Universal Robots PolyScope program: mecspe_refactor.urp

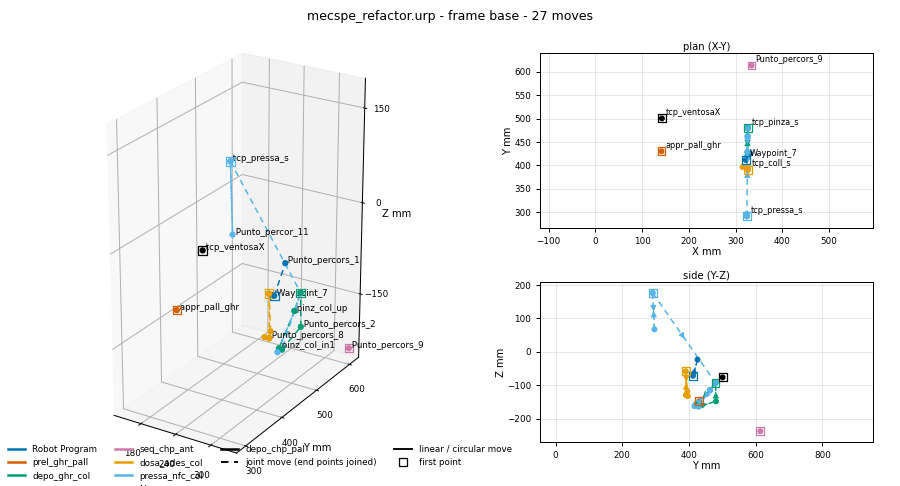
[picture p0: tool path of mecspe_refactor.urp in frame base, 27 of 40 moves have a stored position in this frame; points joined in program order, loops and branches not executed]
Program mecspe_refactor (installation=mecspe_install directory=/home/ur/ursim-current/programs/mecspe2 createdIn=3.15.4.106291 lastSavedIn=3.15.4.106291 robotSerialNumber=2018359999)
Calibrated DH parameters: a=[0.000104, -0.381245, -0.385946, 0.00002, 0.000083, 0]; d=[0.089177, 59.99214, -36.297918, -23.584132, 0.094784, 0.082552]; alpha=[1.570197, -0.003145, 0.002952, 1.570494, -1.570091, 0]; deltaTheta=[-0.00001, -0.459739, 0.638868, -0.17972, -0.000006, -0.000462]
InitVariablesNode variables(variable(name=ghr, expression=2), variable(name=nCycle, expression=0), variable(name=pallStocks, expression=[16,16,16,40,16,16,16,40,16,16,16,40,16,40,0,0,0,0,0,0,0,0,0,0]), variable(name=pick, expression=[0,0]))
BeforeStart
  Script file /home/ur/ursim-current/programs/mecspe2/calc_pose_to_position.script
    | def calc_pose_to_position(pose, feature, position):
    | 
    |    PoseRelativeToFeature = pose_trans(pose_inv(feature), pose)
    | 
    |    diff = pose_sub(position, PoseRelativeToFeature)
    |    vect = p[diff[0], diff[1], diff[2], 0, 0, 0]
    | 
    |    MoveTCPRelativeToFeature = pose_add(PoseRelativeToFeature, vect)
    |    return pose_trans(feature, MoveTCPRelativeToFeature)
    | 
    | end
  Script file /home/ur/ursim-current/programs/mecspe2/calc_item_position.script
    | def calc_item_position(item, prop, grid, module, seat, compens):
    | 
    |     # calcola la posizione assoluta del pezzo scelto da pickPalletItem
    | 
    |     # nPosX è il numero di colonne
    |     # nPosY è il numero di righe
    |     # distX è la distanza tra colonne
    |     # distY è la distanza tra righe
    |     # [posX1, posY1] è la posizione del primo pezzo rispetto all'origine del pallet
    | 
    |     nPallet = module # module e seat partono da 1
    |     nItem = seat
    | 
    |     nPosXgrid = grid[0] # numero di posizioni della giglia in X
    |     distXgrid = grid[2] # distanza tra gli slot della griglia in X
    |     distYgrid = grid[3] # distanza tra gli slot della griglia in Y
    | 
    |     pallPosX = nPallet%nPosXgrid
    |     if(pallPosX==0): pallPosX = nPosXgrid end
    |     pallPosY = ceil(nPallet/nPosXgrid)
    | 
    |     pallPosX1 = grid[4]
    |     pallPosY1 = grid[5]
    | 
    | 
    |     nPosX = prop[item,0]
    |     nPosY = prop[item,1]
    |     distX = prop[item,2]
    |     distY = prop[item,3]
    |     posX1 = prop[item,4]
    |     posY1 = prop[item,5]
    | 
    |     posX = nItem%nPosX
    |     if(posX==0): posX = nPosX end
    |     posY = ceil(nItem/nPosX)
    | 
    |     position = p[0,0,0,0,0,0]
    | 
    |     X=distX*(posX - 1) + posX1 + distXgrid*(pallPosX - 1) + pallPosX1 + compens[0]*1000
    |     Y=distY*(posY - 1) + posY1 + distYgrid*(pallPosY - 1) + pallPosY1 + compens[1]*1000
    | 
    |     position[0] = X/1000
    |     position[1] = Y/1000
    | 
    |     return position
    | 
    |  end
  Script file /home/ur/ursim-current/programs/mecspe2/calc_compens_pos.script
    | def calc_compens_pos(item, prop, grid, module, feature, posAppr):
    | 
    | 	compens = p[0,0,0,0,0,0]
    | 	posPred = calc_item_position(item, prop, grid, module, 1, compens)
    | 
    | 	posApprFeat = pose_trans(pose_inv(feature), posAppr)
    | 	diff = pose_sub(posApprFeat - posPred)
    | 
    | 	compens[0] = diff[0]
    | 	compens[1] = diff[1]
    | 
    | 	return compens
    | 
    | end
  Script file /home/ur/ursim-current/programs/mecspe2/tcpMov.script
    | def tcpMov(vect):
    | 
    |     # FeaturePose is the pose for the feature
    |     # vect = p[0.1, 0, 0, 0, 0, 0] makes us move 10cm in the X direction of the feature
    |     # credits: https://forum.universal-robots.com/t/move-tcp-relative-to-feature/15492
    | 
    |    tcp_pose = get_actual_tcp_pose()
    |    return pose_add(tcp_pose, vect)
    | 
    | 
    | end
  Script file /home/ur/ursim-current/programs/mecspe2/gen_tcp_grid.script
    | def next_tcp_grid_pos(cur_pos,size,dist):
    | 
    | # size e' la dimensione della griglia da generare,
    | # 2 significa 2x2, 3 significa 3x3 etc
    | 
    | rel_p = [0,0]
    | tcpp = get_actual_tcp_pose()
    | 
    | posX = cur_pos%size
    | if(posX==0): posX = size end
    | posY = ceil(cur_pos/size)
    | 
    | actual_dx = -dist*(size-1)/2 + (posX-1)*dist
    | actual_dy= -dist*(size-1)/2 + (posY-1)*dist
    | 
    | posX = (cur_pos+1)%size
    | if(posX==0): posX = size end
    | posY = ceil((cur_pos+1)/size)
    | 
    | next_dx = -dist*(size-1)/2 + (posX-1)*dist
    | next_dy= -dist*(size-1)/2 + (posY-1)*dist
    | 
    | rel_p = [next_dx - actual_dx, next_dy - actual_dy]
    | 
    | return rel_p
    | 
    | end
  Script file /home/ur/ursim-current/programs/andrea11/stockUpdate.script_bak
    | def stockUpdate(pick,stock):
    | 
    |     # simple function that ingests the output of pickItem and returns the
    |     # modified stock array. just so to avoid using global variables and
    |     # multi-dimensional arrays
    | 
    |     i = pick[0]
    |     stock[i] = stock[i] - 1
    |     return stock
    | 
    | 
    | end
  Script file /home/ur/ursim-current/programs/mecspe2/pickPalletItem.script
    | def pickPalletItem(type, pallDefs, pallTypes, pallStocks):
    | 
    |   # seleziona un pezzo sulla griglia, noti il tipo di pezzo e lo stato della griglia
    | 
    |   # lo script funziona finché le variabili del robot non vengono resettate. Tuttavia, anche
    |   # in caso di riavvio, è possibile scrivere manualmente le info sulla griglia e lo stock
    |   # all'inizio del programma, così da 'insegnare' al robot dove farlo
    |   # riprendere
    | 
    |   iPallet = 0 # inizializzo l'id del pallet
    | 
    |   while iPallet < length(pallStocks):
    | 
    |     if pallTypes[iPallet] == type and pallStocks[iPallet] > 0 :
    | 
    |       nItems = pallStocks[iPallet] # numero di pezzi nello stock del pallet iesimo
    | 
    |       nPosX = pallDefs[type,0] # numero di posizioni lungo x, come definito per il pallet di tipo "type"
    |       nPosY = pallDefs[type,1] # numero di posizioni lungo y, come definito per il pallet di tipo "type"
    | 
    |       stockMax = nPosX*nPosY
    |       iItem = stockMax - nItems # id del pezzo
    | 
    |       pick = [iPallet,iItem]
    | 
    |       # pick = [id del pallet, id del pezzo]
    | 
    |       return pick
    |  end
    | iPallet = iPallet + 1
    | end
    | end
  Script file /home/ur/ursim-current/programs/mecspe2/ini_grid.script
    | def ini_grid():
    | 
    |     # grid = [nPallPosX, nPallPosY, distPallX, distPallY, pallPosX1, pallPosY1, pallPosZ1]
    |     # la struttura e' del tutto analoga in logica con quella espressa in defs
    |     grid = [4, 6, 90, 90, 10, 20, 6]
    |     return grid
    | end
  Script file /home/ur/ursim-current/programs/mecspe2/ini_defs.script
    | chp = 1
    | ghr = 2
    | 
    | def ini_defs():
    | 
    |     # definition = [nPosX,nPosY,distX,distY,posX1,posY1,posZ1]
    | 
    |     # nPosX è il numero di colonne
    |     # nPosY è il numero di righe
    |     # distX è la distanza tra colonne
    |     # distY è la distanza tra righe
    |     # [posX1, posY1] è la posizione del primo pezzo rispetto all'origine del pallet
    |     # posZ1 e' la posizione che deve raggiungere il TCP lungo asse Z, che sarebbe asse verticale
    | 
    |     defs = [
    |         [0, 0, 0, 0, 0, 0, 0], # slot vuoto
    |         [4, 10, 18, 8, 17, 10.3, 10], # pallet chip
    |         [4, 4, 21, 21, 12.5, 12.5, 50], # pallet ghiere
    |         [1, 1, 0, 0, 132.06, 44, 16.05], # stazione antenna
    |         [1, 2, 0, 40, 20.256, 24, 27.85], # stazione incollaggio
    |         [1, 1, 0, 0, 40, 40, 50] # cestino
    |     ]
    |     return defs
    | end
  Script file /home/ur/ursim-current/programs/mecspe2/ini_types.script_bak_bak
    | def ini_types():
    | 
    |     visualTypes = [
    | 
    |         [0, 0, 0, 0],
    |         [0, 0, 0, 0],
    |         [0,0,0,0],
    |         [0,0,0,0],
    |         [0,ghr,0,chp],
    |         [0,0,0,0]
    | 
    |     ]
    | 
    | # purtroppo fare questa array vuota di dimensione (righe)x(colonne) per aggirare le limitazioni di UR
    | # bisogna ricordarsi di cambiare questa dichiarazione di types se si cambia dimensione griglia
    | 
    |      types = [0,0,0,0,0,0,0,0,0,0,0,0,0,0,0,0,0,0,0,0,0,0,0,0]
    | 
    |     iii = 0
    |     s = size(visualTypes)
    |     i = 0
    |     while i < s[0]:
    | 
    |         ii=0
    |         while ii < s[1]:
    | 
    |             types[iii] = visualTypes[s[0]-1-i,ii]
    |             ii = ii + 1
    |             iii = iii + 1
    |         end
    |     i = i + 1
    |     end
    |     return types
    | end
  Script file /home/ur/ursim-current/programs/mecspe2/ini_stocks.script
    | def ini_stocks(defs, types):
    | 
    |     global f = -1 # usa questo carattere per inizializzare automaticamente pallet pieni
    | 
    |     visualStocks = [
    | 
    |         [f, f, f, f],
    |         [f, f, f, f],
    |         [f, f, f, f],
    |         [f, f, f, f],
    |         [f, f, f, f],
    |         [f ,f, f, f]
    | 
    |     ]
    | 
    | # purtroppo occorre fare questa array vuota di dimensione (righe)x(colonne) per aggirare le limitazioni di UR
    | # bisogna ricordarsi di cambiare questa dichiarazione di types se si cambia dimensione griglia
    | 
    |      stocks = [0,0,0,0,0,0,0,0,0,0,0,0,0,0,0,0,0,0,0,0,0,0,0,0]
    | 
    |     iii = 0
    |     s = size(visualStocks)
    |     i = 0
    |     while i < s[0]:
    | 
    |         ii=0
    |         while ii < s[1]:
    |             if visualStocks[s[0]-1-i,ii] == f:
    |                 nPosX = defs[types[iii], 0]
    |                 nPosY = defs[types[iii], 1]
    |                 stocks[iii] = nPosX*nPosY
    |             else:
    | 
    |                 stocks[iii] = visualStocks[s[0]-1-i,ii]
    |             end
    |             ii = ii + 1
    |             iii = iii + 1
    |         end
    |     i = i + 1
    |     end
    |     return stocks
    | end
  Script file /home/ur/ursim-current/programs/mecspe2/fun_tens_utensile.script
    | def fun_tens_utensile():
    | 
    | 	i = 0
    | 	# invia 3 "impulsi" alla macchina per assicurarsi che il tool abbia tensione
    | 	while i < 3:
    | 		set_tool_voltage(24)
    | 		sleep(0.24)
    | 		i = i + 1
    | 	end
    | 
    | end
  posApproccio := get_actual_tcp_pose()
  statoPinza := 0
  statoGhiera := 0
  statoChip := 0
  compens := p[0,0,0,0,0,0]
  Set DigitalOutput pin=DO_ventosaOff; digitalValue=1
  Set DigitalOutput pin=DO_ventosaOn; digitalValue=0
  Set DigitalOutput pin=digital_out[2]; digitalValue=0
  pallTypes := ini_types()
  bypassVerifChp := False
  grid := ini_grid()
  pallDefs := ini_defs()
  pallStocks := ini_stocks(pallDefs,pallTypes)
  nCycle := 1
  chp_check := False
  Script: fun_tens_utensile()
  Wait Sleep waitTime=1
Robot Program (runOnlyOnce=false)
  MoveJ speed 60 deg/s, acceleration 80 deg/s^2 (useActiveTCP=true)
    Waypoint Waypoint_7: TCP in base x=321.623 y=412.075 z=-71.725 mm, rx=1.5831 ry=-2.4822 rz=0.1268 rad; joints [-138.339, -65.21, 105.073, -118.045, -93.062, 36.92] deg; flange x=345.08 y=447.244 z=123.756 mm, rx=2.1618 ry=-1.9789 rz=0.0478 rad
  Timer (action=Start) variable(name=timer_1)
  apprendimento := True
  item := ghr
  pick := pickPalletItem(item,pallDefs,pallTypes,pallStocks)
  lastpick := pick
  Call prel_ghr_pall
  statoGhiera := 1
  Call depo_ghr_col
  statoGhiera := 2
  chp_check := False
  Loop While (checkContinuously=false) expression=chp_check≟ False
    item := chp
    pick := pickPalletItem(item,pallDefs,pallTypes,pallStocks)
    Call prel_chp_pall
    statoChip := 1
    pallStocks := stockUpdate(pick,pallStocks)
    MoveJ speed 60 deg/s, acceleration 80 deg/s^2 (useActiveTCP=false) tcp=Ventosa
      Waypoint Punto_percors_1: TCP in base x=331.541 y=425.449 z=-23.301 mm, rx=1.7621 ry=-0.7398 rz=-1.7726 rad; joints [-145.076, -38.163, 77.174, -38.938, -53.96, -45.259] deg; flange x=377.019 y=458.221 z=10.448 mm, rx=1.7621 ry=-0.7398 rz=-1.7726 rad
    Call seq_chp_ant
    If chp_check≟ True
      Call dosa_ades_col
      Call pressa_nfc_col
      Call prel_ghr_col
    Else 
      Call depo_chp_pal
Thread Thread_1 (runOnlyOnce=false)
  If timer_1>4
    Timer (action=Reset) variable=timer_1
    Script: fun_tens_utensile()
    Timer (action=Start) variable=timer_1
SubProgram -> prel_ghr_pall
SubProgram  [hidden by the author, left out]
SubProgram  [hidden by the author, left out]
SubProgram depo_ghr_pall [hidden by the author, left out]
SubProgram -> depo_chp_pal
SubProgram -> seq_chp_ant
SubProgram -> depo_ghr_col
SubProgram -> dosa_ades_col
SubProgram -> pressa_nfc_col
SubProgram prel_ghr_pall (keepSynchronizedWithDisk=false)
  If apprendimento≟ True
    MoveJ speed 60 deg/s, acceleration 80 deg/s^2 (useActiveTCP=false) tcp=Pinza
      Waypoint appr_pall_ghr: TCP in base x=141.508 y=430.186 z=-147.75 mm, rx=0.607 ry=-1.4882 rz=-0.6293 rad; joints [-125.755, -39.244, 81.167, -41.963, -34.571, 44.831] deg; flange x=189.515 y=570.182 z=1.456 mm, rx=0.607 ry=-1.4882 rz=-0.6293 rad
      modulo :=  (valueSource=Operator message=Specificare il numero di modulo usato per l'apprendimento valueType=Integer)
  Else 
    MoveJ speed 60 deg/s, acceleration 80 deg/s^2 (useActiveTCP=false) tcp=Pinza
      Script: posApproccio = pose_trasf(posa, riferimento, vettore)
      Waypoint Waypoint (Variable): variable=posApproccio
  MoveL speed 250 mm/s, acceleration 1200 mm/s^2 (useActiveTCP=false) tcp=Pinza; feature=Base
    Waypoint Waypoint_1 (Relative): relativeFromPosition TCP in base x=143.961 y=537.139 z=34.835 mm, rx=0.607 ry=-1.4882 rz=-0.6293 rad; joints [-125.506, -39.287, 81.209, -42.035, -34.619, 44.824] deg; TCP in base x=143.457 y=501.955 z=-0.687 mm, rx=0.607 ry=-1.4882 rz=-0.6293 rad; joints [-127.449, -38.931, 87.822, -48.999, -36.562, 44.817] deg; flange x=189.012 y=534.998 z=-34.066 mm, rx=0.607 ry=-1.4882 rz=-0.6293 rad
  MoveL speed 50 mm/s, acceleration 100 mm/s^2 (useActiveTCP=false) tcp=Pinza; feature=Base
    Waypoint Waypoint_2 (Relative): relativeFromPosition TCP in base x=143.457 y=501.955 z=-0.687 mm, rx=0.607 ry=-1.4882 rz=-0.6293 rad; joints [-127.449, -38.931, 87.822, -48.999, -36.562, 44.817] deg; TCP in base x=143.286 y=489.992 z=-12.765 mm, rx=0.607 ry=-1.4882 rz=-0.6293 rad; joints [-128.156, -38.626, 89.864, -51.344, -37.269, 44.815] deg; flange x=188.841 y=523.035 z=-46.144 mm, rx=0.607 ry=-1.4882 rz=-0.6293 rad
    SuppressedNode
      Script: tool()
    Waypoint Waypoint_3 (Relative): relativeFromPosition TCP in base x=143.286 y=489.992 z=-12.765 mm, rx=0.607 ry=-1.4882 rz=-0.6293 rad; joints [-128.156, -38.626, 89.864, -51.344, -37.269, 44.815] deg; TCP in base x=143.457 y=501.955 z=-0.687 mm, rx=0.607 ry=-1.4882 rz=-0.6293 rad; joints [-127.449, -38.931, 87.822, -48.999, -36.562, 44.817] deg; flange x=189.012 y=534.998 z=-34.066 mm, rx=0.607 ry=-1.4882 rz=-0.6293 rad
  MoveL speed 250 mm/s, acceleration 1200 mm/s^2 (useActiveTCP=false) tcp=Pinza; feature=Base
    Waypoint Waypoint_4 (Relative): relativeFromPosition TCP in base x=143.457 y=501.955 z=-0.687 mm, rx=0.607 ry=-1.4882 rz=-0.6293 rad; joints [-127.449, -38.931, 87.822, -48.999, -36.562, 44.817] deg; TCP in base x=143.961 y=537.139 z=34.835 mm, rx=0.607 ry=-1.4882 rz=-0.6293 rad; joints [-125.506, -39.287, 81.209, -42.035, -34.619, 44.824] deg; flange x=189.515 y=570.182 z=1.456 mm, rx=0.607 ry=-1.4882 rz=-0.6293 rad
SubProgram depo_ghr_col (keepSynchronizedWithDisk=false)
  MoveJ speed 60 deg/s, acceleration 80 deg/s^2 (useActiveTCP=false) tcp=Pinza
    Waypoint tcp_pinza_s: TCP in base x=326.011 y=479.267 z=-92.696 mm, rx=0.6076 ry=-1.4868 rz=-0.6287 rad; joints [-134.797, -24.75, 41.969, -17.153, -43.759, 44.739] deg; flange x=373.998 y=619.302 z=56.479 mm, rx=0.6076 ry=-1.4868 rz=-0.6287 rad
    Waypoint pinz_col_up: TCP in base x=325.773 y=462.541 z=-115.349 mm, rx=-0.2128 ry=-1.5595 rz=0.1908 rad; joints [-132.675, 4.221, 14.51, -18.717, -41.716, 104.821] deg; flange x=376.545 y=660.076 z=-162.724 mm, rx=-0.2162 ry=-1.5589 rz=0.1901 rad
    Waypoint pinz_col_in1: TCP in base x=325.228 y=420.094 z=-158.165 mm, rx=-0.2127 ry=-1.5596 rz=0.1906 rad; joints [-134.83, -0.501, 31.804, -31.303, -43.826, 104.834] deg; flange x=374.048 y=618.963 z=-205.428 mm, rx=-0.2127 ry=-1.5596 rz=0.1906 rad
    SuppressedNode
      URCap Close Gripper (SCHUNK End-of-Arm Modular System for UR, SCHUNK GmbH & Co.)
    Waypoint pinz_col_out: TCP in base x=325.373 y=428.559 z=-163.725 mm, rx=-0.2126 ry=-1.5596 rz=0.1907 rad; joints [-134.386, 1.907, 27.313, -29.22, -43.4, 104.831] deg; flange x=374.171 y=627.435 z=-210.98 mm, rx=-0.2126 ry=-1.5596 rz=0.1907 rad
    SuppressedNode
      Waypoint pinz_col_up: TCP in base x=353.537 y=408.471 z=-60.29 mm, rx=1.9378 ry=-1.1643 rz=-1.0825 rad; joints [-133.591, -22.853, 54.464, -66.388, -55.09, 0.038] deg; flange x=383.886 y=633.812 z=-67.559 mm, rx=1.9378 ry=-1.1643 rz=-1.0825 rad
    Waypoint Punto_percors_2: TCP in base x=326.04 y=480.901 z=-148.453 mm, rx=0.4029 ry=-1.5348 rz=-0.4259 rad; joints [-133.017, -11.499, 29.335, -17.8, -41.967, 59.778] deg; flange x=376.733 y=653.438 z=-40.877 mm, rx=0.3991 ry=-1.5354 rz=-0.4274 rad
    SuppressedNode
      URCap Open Gripper (SCHUNK End-of-Arm Modular System for UR, SCHUNK GmbH & Co.)
    Waypoint tcp_pinza_s: TCP in base x=326.011 y=479.267 z=-92.696 mm, rx=0.6076 ry=-1.4868 rz=-0.6287 rad; joints [-134.797, -24.75, 41.969, -17.153, -43.759, 44.739] deg; flange x=373.998 y=619.302 z=56.479 mm, rx=0.6076 ry=-1.4868 rz=-0.6287 rad
SubProgram prel_chp_pall [hidden by the author, left out]
SubProgram seq_chp_ant (keepSynchronizedWithDisk=false)
  If apprendimento≟ True
    MoveJ speed 60 deg/s, acceleration 80 deg/s^2 (useActiveTCP=false) tcp=Ventosa
      Waypoint Punto_percors_9: TCP in base x=334.202 y=613.623 z=-237.914 mm, rx=1.7619 ry=-0.7398 rz=-1.7727 rad; joints [-133.692, 7.188, 14.603, -21.767, -42.719, -45.183] deg; flange x=379.684 y=646.401 z=-204.176 mm, rx=1.7619 ry=-0.7398 rz=-1.7727 rad
  Else 
    MoveJ speed 60 deg/s, acceleration 80 deg/s^2 (useActiveTCP=false) tcp=Pinza
      SuppressedNode
        Script: pos_approccio = calc_rel_pose()
      Waypoint Waypoint (Variable): variable=posApproccio
  MoveL speed 50 mm/s, acceleration 100 mm/s^2 (useActiveTCP=false) tcp=Ventosa; feature=Base
    Waypoint Waypoint_5 (Relative): relativeFromPosition TCP in base x=334.202 y=613.623 z=-237.914 mm, rx=1.7619 ry=-0.7398 rz=-1.7727 rad; joints [-133.509, 7.247, 14.462, -21.694, -42.684, -45.282] deg; TCP in base x=333.934 y=593.03 z=-258.697 mm, rx=1.762 ry=-0.7397 rz=-1.7726 rad; joints [-134.549, 4.522, 23.777, -28.293, -43.727, -45.281] deg; flange x=379.412 y=625.807 z=-224.951 mm, rx=1.762 ry=-0.7397 rz=-1.7726 rad
    If bypassVerifChp≟ True
      chp_check := True
    ElseIf digital_in[0]≟ False
      chp_check :=  (valueSource=Operator message=L'antenna nfc non risponde. Si prega di confermare la funzionalita' del sensore valueType=Boolean)
    Else 
      Loop Counting (count=5) loopVariable(name=Loop_1)
        Wait Sleep waitTime=0.5
        If DI_chpVerif≟ True
          chp_check := True
    Waypoint Waypoint_6 (Relative): relativeFromPosition TCP in base x=333.934 y=593.03 z=-258.697 mm, rx=1.762 ry=-0.7397 rz=-1.7726 rad; joints [-134.549, 4.522, 23.777, -28.293, -43.727, -45.281] deg; TCP in base x=334.202 y=613.623 z=-237.914 mm, rx=1.7619 ry=-0.7398 rz=-1.7727 rad; joints [-133.509, 7.247, 14.462, -21.694, -42.684, -45.282] deg; flange x=379.684 y=646.401 z=-204.176 mm, rx=1.7619 ry=-0.7398 rz=-1.7727 rad
SubProgram dosa_ades_col (keepSynchronizedWithDisk=false)
  MoveJ speed 60 deg/s, acceleration 80 deg/s^2 (useActiveTCP=false) tcp=Dosatore_Colla
    Waypoint tcp_coll_s: TCP in base x=326.049 y=390.336 z=-58.733 mm, rx=1.5073 ry=-2.6452 rz=0.2028 rad; joints [-138.926, -70.014, 111.07, -124.336, -96.301, 42.443] deg; flange x=328.586 y=422.248 z=138.688 mm, rx=2.1203 ry=-2.1445 rz=0.1587 rad
    Waypoint Punto_percors_7: TCP in base x=326.117 y=395.016 z=-120.075 mm, rx=1.5072 ry=-2.6453 rz=0.2028 rad; joints [-138.56, -63.27, 112.967, -132.934, -96.298, 42.835] deg; flange x=328.653 y=426.927 z=77.346 mm, rx=2.1202 ry=-2.1446 rz=0.1587 rad
    Waypoint Punto_percors_8: TCP in base x=326.087 y=391.561 z=-129.594 mm, rx=1.5073 ry=-2.6453 rz=0.2028 rad; joints [-138.834, -62.452, 113.712, -134.529, -96.337, 42.56] deg; flange x=328.619 y=423.469 z=67.828 mm, rx=2.1203 ry=-2.1446 rz=0.1587 rad
  MoveL speed 250 mm/s, acceleration 1200 mm/s^2 (useActiveTCP=false) tcp=Dosatore_Colla; feature=Base
    Waypoint Punto_percors_8: TCP in base x=326.087 y=391.561 z=-129.594 mm, rx=1.5073 ry=-2.6453 rz=0.2028 rad; joints [-138.834, -62.452, 113.712, -134.529, -96.337, 42.56] deg; flange x=328.619 y=423.469 z=67.828 mm, rx=2.1203 ry=-2.1446 rz=0.1587 rad
    Waypoint arco01: TCP in base x=314.98 y=396.61 z=-132.865 mm, rx=-1.4222 ry=2.3645 rz=-0.9681 rad; joints [-120.617, -54.723, 114.843, -141.201, -129.749, 60.945] deg; flange x=216.441 y=481.445 z=19.098 mm, rx=-2.0946 ry=2.021 rz=-1.0736 rad
    Set DigitalOutput pin=digital_out[2]; digitalValue=1
    Wait Sleep waitTime=0.5
    Waypoint Punto_percors_8: TCP in base x=326.087 y=391.561 z=-129.594 mm, rx=1.5073 ry=-2.6453 rz=0.2028 rad; joints [-138.834, -62.452, 113.712, -134.529, -96.337, 42.56] deg; flange x=328.619 y=423.469 z=67.828 mm, rx=2.1203 ry=-2.1446 rz=0.1587 rad
    Set DigitalOutput pin=digital_out[2]; digitalValue=0
  MoveJ speed 60 deg/s, acceleration 80 deg/s^2 (useActiveTCP=false) tcp=Dosatore_Colla
    Waypoint tcp_coll_s: motionParameters(blendRadius=0.005); TCP in base x=326.049 y=390.336 z=-58.733 mm, rx=1.5073 ry=-2.6452 rz=0.2028 rad; joints [-138.926, -70.014, 111.07, -124.336, -96.301, 42.443] deg; flange x=328.586 y=422.248 z=138.688 mm, rx=2.1203 ry=-2.1445 rz=0.1587 rad
SubProgram pressa_nfc_col (keepSynchronizedWithDisk=false)
  MoveJ speed 60 deg/s, acceleration 80 deg/s^2 (useActiveTCP=false) tcp=Pressa
    SuppressedNode
      Waypoint tcp_ventosaY_s: TCP in base x=355.984 y=389.916 z=-58.857 mm, rx=-1.401 ry=-1.0647 rz=1.3858 rad; joints [-146.472, -36.177, 73.345, -37.097, -55.375, 194.745] deg; flange x=401.93 y=456.119 z=8.64 mm, rx=-1.401 ry=-1.0647 rz=1.3858 rad
    Waypoint tcp_pressa_s: TCP in base x=324.299 y=291.031 z=176.511 mm, rx=-1.4012 ry=-1.0643 rz=1.3857 rad; joints [-148.69, -46.659, 85.022, -38.277, -57.561, -165.274] deg; flange x=370.992 y=407.578 z=60.385 mm, rx=-1.4012 ry=-1.0643 rz=1.3857 rad
    Waypoint Punto_percor_11: TCP in base x=324.225 y=296.228 z=67.341 mm, rx=-1.3969 ry=-1.0517 rz=1.3843 rad; joints [-148.364, -36.011, 84.683, -48.026, -56.743, -165.537] deg; flange x=370.899 y=412.4 z=-49.168 mm, rx=-1.3969 ry=-1.0517 rz=1.3843 rad
    Wait Sleep waitTime=5
    Waypoint tcp_pressa_s: TCP in base x=324.299 y=291.031 z=176.511 mm, rx=-1.4012 ry=-1.0643 rz=1.3857 rad; joints [-148.69, -46.659, 85.022, -38.277, -57.561, -165.274] deg; flange x=370.992 y=407.578 z=60.385 mm, rx=-1.4012 ry=-1.0643 rz=1.3857 rad
  MoveJ speed 60 deg/s, acceleration 80 deg/s^2 (useActiveTCP=false) tcp=Pinza
    Waypoint tcp_pinza_s: TCP in base x=326.011 y=479.267 z=-92.696 mm, rx=0.6076 ry=-1.4868 rz=-0.6287 rad; joints [-134.797, -24.75, 41.969, -17.153, -43.759, 44.739] deg; flange x=373.998 y=619.302 z=56.479 mm, rx=0.6076 ry=-1.4868 rz=-0.6287 rad
    Waypoint pinz_col_up: TCP in base x=325.773 y=462.541 z=-115.349 mm, rx=-0.2128 ry=-1.5595 rz=0.1908 rad; joints [-132.675, 4.221, 14.51, -18.717, -41.716, 104.821] deg; flange x=376.545 y=660.076 z=-162.724 mm, rx=-0.2162 ry=-1.5589 rz=0.1901 rad
    Waypoint pinz_col_out: TCP in base x=325.373 y=428.559 z=-163.725 mm, rx=-0.2126 ry=-1.5596 rz=0.1907 rad; joints [-134.386, 1.907, 27.313, -29.22, -43.4, 104.831] deg; flange x=374.171 y=627.435 z=-210.98 mm, rx=-0.2126 ry=-1.5596 rz=0.1907 rad
    Waypoint pinz_col_in: TCP in base x=325.232 y=416.122 z=-162.784 mm, rx=-0.2125 ry=-1.5596 rz=0.1904 rad; joints [-135.043, -0.583, 32.776, -32.194, -44.036, 104.821] deg; flange x=374.053 y=615.003 z=-209.997 mm, rx=-0.2125 ry=-1.5596 rz=0.1904 rad
    SuppressedNode
      URCap Open Gripper (SCHUNK End-of-Arm Modular System for UR, SCHUNK GmbH & Co.)
    Waypoint pinz_col_up: TCP in base x=325.773 y=462.541 z=-115.349 mm, rx=-0.2128 ry=-1.5595 rz=0.1908 rad; joints [-132.675, 4.221, 14.51, -18.717, -41.716, 104.821] deg; flange x=376.545 y=660.076 z=-162.724 mm, rx=-0.2162 ry=-1.5589 rz=0.1901 rad
    SuppressedNode
      Waypoint pinz_col_up: TCP in base x=353.537 y=408.471 z=-60.29 mm, rx=1.9378 ry=-1.1643 rz=-1.0825 rad; joints [-133.591, -22.853, 54.464, -66.388, -55.09, 0.038] deg; flange x=383.886 y=633.812 z=-67.559 mm, rx=1.9378 ry=-1.1643 rz=-1.0825 rad
    SuppressedNode
      Waypoint Punto_percors_2: TCP in base x=354.064 y=441.822 z=-77.166 mm, rx=1.8482 ry=-1.2116 rz=-0.904 rad; joints [-131.419, -13.619, 42.947, -63.355, -59.194, 8.709] deg; flange x=380.052 y=663.563 z=-120.852 mm, rx=1.8482 ry=-1.2116 rz=-0.904 rad
    SuppressedNode
      URCap Open Gripper (SCHUNK End-of-Arm Modular System for UR, SCHUNK GmbH & Co.)
    Waypoint tcp_pinza_s: TCP in base x=326.011 y=479.267 z=-92.696 mm, rx=0.6076 ry=-1.4868 rz=-0.6287 rad; joints [-134.797, -24.75, 41.969, -17.153, -43.759, 44.739] deg; flange x=373.998 y=619.302 z=56.479 mm, rx=0.6076 ry=-1.4868 rz=-0.6287 rad
SubProgram prel_ghr_col [hidden by the author, left out]
SubProgram depo_chp_pal (keepSynchronizedWithDisk=false)
  If apprendimento≟ True
    MoveJ speed 60 deg/s, acceleration 80 deg/s^2 (useActiveTCP=false) tcp=Ventosa
      Waypoint tcp_ventosaX: TCP in base x=142.442 y=500.567 z=-76.685 mm, rx=1.7622 ry=-0.7397 rz=-1.7725 rad; joints [-127.721, -38.126, 88.043, -49.879, -36.592, -45.229] deg; flange x=187.914 y=533.343 z=-42.931 mm, rx=1.7622 ry=-0.7397 rz=-1.7725 rad
  Else 
    MoveJ speed 60 deg/s, acceleration 80 deg/s^2 (useActiveTCP=false) tcp=Pinza
      SuppressedNode
        Script: pos_approccio = calc_rel_pose()
      Waypoint Waypoint (Variable): variable=posApproccio
  MoveL speed 250 mm/s, acceleration 1000 mm/s^2 (useActiveTCP=false) tcp=Ventosa; feature=Base
    Waypoint Punto_percor_22 (Relative): relativeFromPosition TCP in base x=35.118 y=689.646 z=-262.532 mm, rx=1.7853 ry=-0.7339 rz=-1.771 rad; joints [-111.426, -3.8, 43.305, -41.846, -20.436, -43.809] deg; TCP in base x=33.407 y=563.018 z=-390.38 mm, rx=1.7855 ry=-0.7339 rz=-1.7712 rad; joints [-115.654, -0.107, 63.287, -65.282, -24.633, -44.07] deg; flange x=78.389 y=595.329 z=-355.54 mm, rx=1.7855 ry=-0.7339 rz=-1.7712 rad
  MoveL speed 100 mm/s, acceleration 100 mm/s^2 (useActiveTCP=false) tcp=Ventosa; feature=Base
    Set DigitalOutput pin=DO_ventosaOff; digitalValue=1
    Set DigitalOutput pin=digital_out[0]; digitalValue=0
    Waypoint Punto_percor_24 (Relative): relativeFromPosition TCP in base x=33.415 y=563.017 z=-390.376 mm, rx=1.7855 ry=-0.7339 rz=-1.7712 rad; joints [-115.654, -0.107, 63.287, -65.283, -24.634, -44.07] deg; TCP in base x=33.33 y=555.287 z=-398.137 mm, rx=1.7856 ry=-0.7338 rz=-1.7712 rad; joints [-115.969, 0.436, 63.978, -66.501, -24.949, -44.093] deg; flange x=78.312 y=587.594 z=-363.292 mm, rx=1.7856 ry=-0.7338 rz=-1.7712 rad
    Wait Sleep waitTime=2
    Waypoint Punto_percor_25 (Relative): relativeFromPosition TCP in base x=33.325 y=555.289 z=-398.147 mm, rx=1.7856 ry=-0.7337 rz=-1.7712 rad; joints [-115.968, 0.437, 63.976, -66.502, -24.954, -44.093] deg; TCP in base x=33.499 y=565.846 z=-387.472 mm, rx=1.7856 ry=-0.7336 rz=-1.7711 rad; joints [-115.544, -0.308, 63.029, -64.836, -24.533, -44.068] deg; flange x=78.474 y=598.159 z=-352.623 mm, rx=1.7856 ry=-0.7336 rz=-1.7711 rad
  MoveL speed 250 mm/s, acceleration 1200 mm/s^2 (useActiveTCP=false) tcp=Ventosa; feature=Base
    Waypoint Punto_percor_26 (Relative): relativeFromPosition TCP in base x=33.484 y=565.888 z=-387.462 mm, rx=1.7857 ry=-0.7336 rz=-1.7712 rad; joints [-115.542, -0.308, 63.027, -64.836, -24.525, -44.07] deg; TCP in base x=35.22 y=689.62 z=-262.535 mm, rx=1.7855 ry=-0.7337 rz=-1.7711 rad; joints [-111.434, -3.807, 43.319, -41.865, -20.444, -43.812] deg; flange x=80.197 y=721.935 z=-227.692 mm, rx=1.7855 ry=-0.7337 rz=-1.7711 rad
